SYSTEM ModLib (* Library only; the modules' systems use these types *)
  (* Standard: 61499-2 *)
  DEVICE FORTE_PC : iec61499::system::FORTE_PC(MGR_ID := "localhost:61499")
    {SET_ATTRIBUTE(Profile, HOLOBLOC)} (* device profile *)
    RESOURCE RES : iec61499::system::EMB_RES
    END_RESOURCE
  END_DEVICE
END_SYSTEM
